// TIA Portal V15 export
// export: Created 2019-01-11T14:30:54.9334832Z, ExportSetting WithDefaults, WithReadOnly, DisplayName Totally Integrated Automation Portal, DisplayVersion V15 Update 2, DisplayName TIA Portal Openness, DisplayVersion V15 Update 2, DisplayName STEP 7 Professional, DisplayVersion V15 Update 2, DisplayName STEP 7 Safety, DisplayVersion V15, DisplayName WinCC Professional, DisplayVersion V15 Update 2, DisplayName SIMATIC Visualization Architect, DisplayVersion V15 Update 1
FUNCTION "SEQUENCENAME_Call" : Void   // FC63, FBD
TITLE = SEQUENCENAME Station 30 sequence / SEQUENCENAME Station 30 Ablaufkette
{ S7_Optimized_Access := 'FALSE' }
VERSION : 0.1
// stored: AutoNumber true, CodeModifiedDate 2018-01-29T16:41:56.3122589Z, CompileDate 2018-02-20T10:24:53.0332673Z, CreationDate 2016-05-29T13:51:21.5311573Z, HandleErrorsWithinBlock false, InterfaceModifiedDate 2017-06-29T05:21:04.5631729Z, IsConsistent true, IsIECCheckEnabled false, IsKnowHowProtected false, IsWriteProtected false, LibraryConformanceStatus Error: The block contains calls of single instances. Warning: The object contains access to global data blocks. Warning: The block contains direct access to inputs, outputs, bit memories, indirect access to the registry or indirect access to external memory areas that are unknown at the time of compilation., ModifiedDate 2018-01-29T16:41:56.3122589Z, ParameterModified 2017-06-29T05:21:04.5631728Z, PLCSimAdvancedSupport false, SetENOAutomatically False, StructureModified 2017-06-29T05:21:04.5631729Z, UDAEnableTagReadback false
BEGIN

REGION Network 1: Safety stop OK, provide general enables here / Sicherheitshalt OK, hier allgemeine Freigaben vorsehen
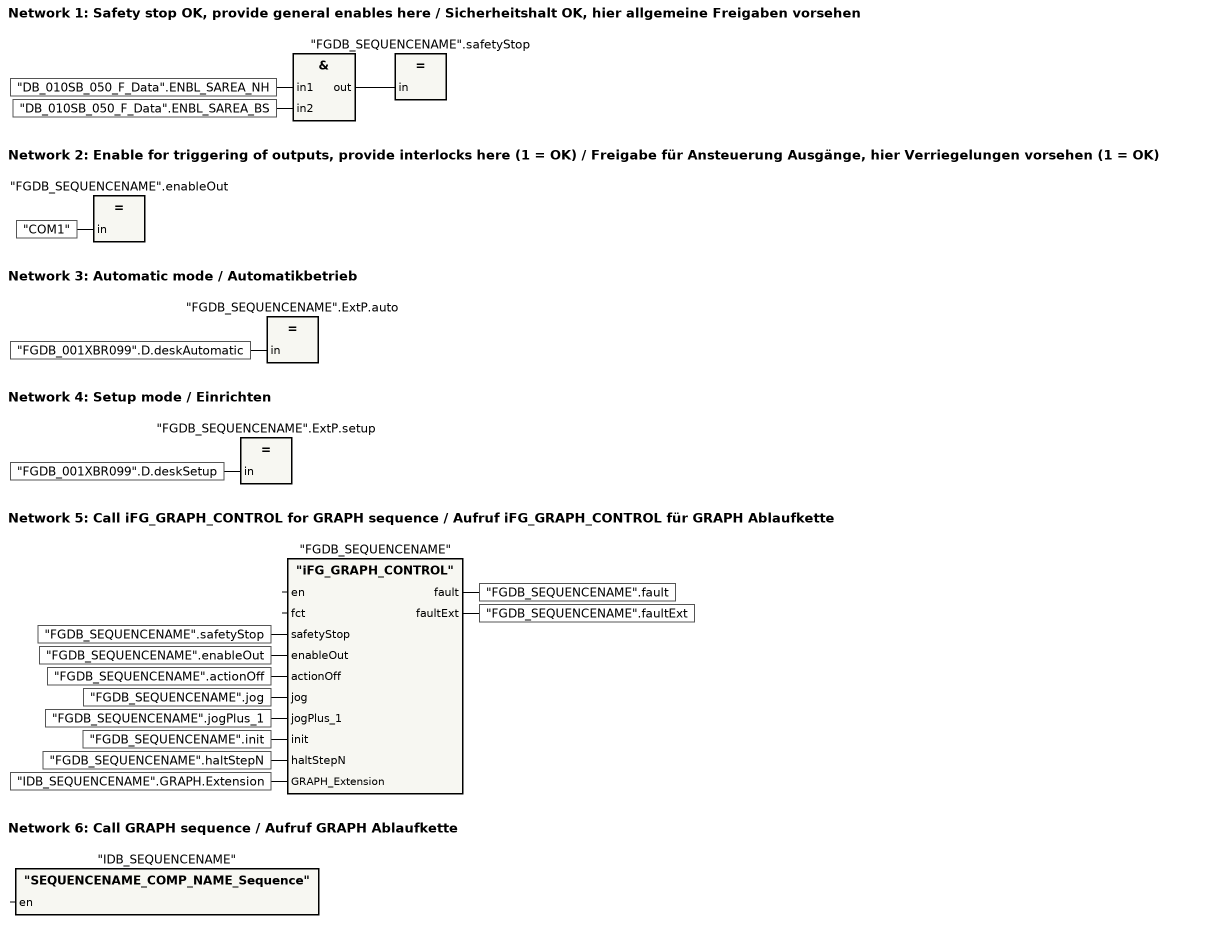
   "FGDB_SEQUENCENAME".safetyStop := "DB_010SB_050_F_Data".ENBL_SAREA_NH AND "DB_010SB_050_F_Data".ENBL_SAREA_BS;
END_REGION

REGION Network 2: Enable for triggering of outputs, provide interlocks here (1 = OK) / Freigabe für Ansteuerung Ausgänge, hier Verriegelungen vorsehen (1 = OK)
   "FGDB_SEQUENCENAME".enableOut := "COM1";
END_REGION

REGION Network 3: Automatic mode / Automatikbetrieb
   "FGDB_SEQUENCENAME".ExtP.auto := "FGDB_001XBR099".D.deskAutomatic;
END_REGION

REGION Network 4: Setup mode / Einrichten
   "FGDB_SEQUENCENAME".ExtP.setup := "FGDB_001XBR099".D.deskSetup;
END_REGION

REGION Network 5: Call iFG_GRAPH_CONTROL for GRAPH sequence / Aufruf iFG_GRAPH_CONTROL für GRAPH Ablaufkette
   "FGDB_SEQUENCENAME"(safetyStop := "FGDB_SEQUENCENAME".safetyStop,   // "iFG_GRAPH_CONTROL"
                       enableOut := "FGDB_SEQUENCENAME".enableOut,
                       actionOff := "FGDB_SEQUENCENAME".actionOff,
                       jog := "FGDB_SEQUENCENAME".jog,
                       jogPlus_1 := "FGDB_SEQUENCENAME".jogPlus_1,
                       init := "FGDB_SEQUENCENAME".init,
                       haltStepN := "FGDB_SEQUENCENAME".haltStepN,
                       GRAPH_Extension := "IDB_SEQUENCENAME".GRAPH.Extension,
                       fault => "FGDB_SEQUENCENAME".fault,
                       faultExt => "FGDB_SEQUENCENAME".faultExt);
END_REGION

REGION Network 6: Call GRAPH sequence / Aufruf GRAPH Ablaufkette
   "IDB_SEQUENCENAME"();   // "SEQUENCENAME_COMP_NAME_Sequence"
END_REGION
END_FUNCTION
